VAR_GLOBAL CONSTANT
	MAX_CSV_ROWS 			: UDINT := 512; (*gc.uiMaxNrOfDMXChannel*)
	MAX_CSV_COLUMNS 		: UDINT := 2;
	MAX_CSV_FIELD_LENGTH	: UDINT := 4;
END_VAR

(* stored: Version 1.1.0.1, ProductVersion 3.1.4024.6
   GVL GVL: Id {44469a28-03d3-42b1-b274-3d87aae2f87d} *)
